INTERFACE I_ReportGenerator

METHOD PUBLIC Generate
VAR_INPUT
	SourceData : ANY;
	TemplateName : T_MAXSTRING;
	FileName : T_MAXSTRING;
	FilePath : T_MAXSTRING;
END_VAR
END_METHOD

END_INTERFACE

(* stored: Version 1.1.0.1, ProductVersion 3.1.4024.12
   Itf I_ReportGenerator: Id {dac13197-b79f-445b-883b-d6ebecc14a5f}
   Method Generate: Id {c75376d8-1bdf-4cd3-bfa6-9b18d3209753} *)
